# EPICS autosave request: CARSApp/Db/Fluke_settings.req
# FILE... Fluke_settings.req
$(P)$(R)_Init.AOUT
$(P)$(R)_Read.SCAN
file "scalcout_settings.req", P=$(P)$(R)_Convert
file "scalcout_settings.req", P=$(P)$(R)_Calc
